(* IEC 61131-3 sources: PLC_Hydraulic_Press_Control_System/rushi_hydraulic_press/build, 2 files *)

(* ---- plc.st ---- *)
TYPE
  LOGLEVEL : (CRITICAL, WARNING, INFO, DEBUG) := INFO;
END_TYPE

FUNCTION_BLOCK LOGGER
  VAR_INPUT
    TRIG : BOOL;
    MSG : STRING;
    LEVEL : LOGLEVEL := INFO;
  END_VAR
  VAR
    TRIG0 : BOOL;
  END_VAR

  IF TRIG AND NOT TRIG0 THEN
  {{
   LogMessage(GetFbVar(LEVEL),(char*)GetFbVar(MSG, .body),GetFbVar(MSG, .len));
  }}
  END_IF;
  TRIG0:=TRIG;
END_FUNCTION_BLOCK

PROGRAM program0
  VAR
    Start : BOOL;
    Stop : BOOL;
    M_0 : BOOL;
    Press_A : BOOL;
    Press_B : BOOL;
    Press_C : BOOL;
    TON0 : TON;
    TON1 : TON;
    TON2 : TON;
  END_VAR

  M_0 := NOT(Stop) AND (M_0 OR Start);
  TON0(IN := M_0, PT := T#5s);
  Press_A := TON0.Q;
  TON1(IN := M_0, PT := T#7s);
  Press_B := TON1.Q;
  TON2(IN := M_0, PT := T#10s);
  Press_C := TON2.Q;
END_PROGRAM

CONFIGURATION Config0

  RESOURCE Res0 ON PLC
    TASK task0(INTERVAL := T#20ms,PRIORITY := 0);
    PROGRAM instance0 WITH task0 : program0;
  END_RESOURCE
END_CONFIGURATION

(* ---- generated_plc.st ---- *)
PROGRAM program0
  VAR
    Start : BOOL;
    Stop : BOOL;
    M_0 : BOOL;
    Press_A : BOOL;
    Press_B : BOOL;
    Press_C : BOOL;
    TON0 : TON;
    TON1 : TON;
    TON2 : TON;
  END_VAR

  M_0 := NOT(Stop) AND (M_0 OR Start);
  TON0(IN := M_0, PT := T#5s);
  Press_A := TON0.Q;
  TON1(IN := M_0, PT := T#7s);
  Press_B := TON1.Q;
  TON2(IN := M_0, PT := T#10s);
  Press_C := TON2.Q;
END_PROGRAM

CONFIGURATION Config0

  RESOURCE Res0 ON PLC
    TASK task0(INTERVAL := T#20ms,PRIORITY := 0);
    PROGRAM instance0 WITH task0 : program0;
  END_RESOURCE
END_CONFIGURATION
